(* PLC project contactor, Dassault Systèmes ControlBuild 2024x *)
(* stored: creationDateTime 2023-10-03T11:13:14-01:00 *)

(* This module simulates the interlocking of a contactor. It returns its state and a contactor feed-back. *)
FUNCTION_BLOCK equipment_library.contactor
  VAR_INPUT
    voltage380 : BOOL := true;
    cmdSupply : BOOL := true;
    sensorSupply : BOOL := true;
  END_VAR
  VAR_INPUT
    forward : BOOL := false;
  END_VAR
  VAR_OUTPUT
    forwardState : BOOL := false;
  END_VAR
  VAR_OUTPUT
    contactorFB : BOOL := false;
    thermal : BOOL := true;
  END_VAR
  VAR
    memoForward : BOOL := false;
  END_VAR
  VAR CONSTANT
    forwardLogic : BOOL := true;
    thermalLogic : BOOL := false;
  END_VAR
  VAR
    d_forward : BOOL := false;
    v_d_forward : BOOL := false;
    d_electrical : BOOL := false;
    v_d_electrical : BOOL := false;
  END_VAR


ACTION C_source_code:
/* ----------------------------------------------------------------	*/
/* Type : Model of Operative Behaviour					*/
/* Category :  Pre-actuators						*/
/* Author : Dassault Systemes						*/
/* Update date : June 2018							*/
/* ----------------------------------------------------------------	*/
/* This module simulates the interlocking of a contactor.  		*/
/* It returns its state and a contactor feed-back.			*/
/* ----------------------------------------------------------------	*/

/* ----------------------------------------------------------------	*/
/* Management of orders from Control Part					*/
/*	if there is no power supply for command 				*/
/*         the contactor doesn't understand the control order		*/
/* ----------------------------------------------------------------	*/
memoForward=forward & cmdSupply & ! d_electrical;

/* ----------------------------------------------------------------	*/
/* Calculation of the on-state of contactor				*/
/* ----------------------------------------------------------------	*/
forwardState=memoForward & voltage380;

/* ----------------------------------------------------------------	*/
/* Management of the thermal feed-back					*/
/* ----------------------------------------------------------------	*/
if (d_electrical) thermal = v_d_electrical;
else
	thermal = ! thermalLogic & sensorSupply;

/* ----------------------------------------------------------------	*/
/* Management of feedback to Control Part					*/
/*     if a fault is required, the contactor feed-back 		*/
/*		 takes a preset state.					*/
/*	if there is no power supply for sensor 				*/
/*         contactor feed-back returns nothing				*/
/*     else contactor feed-back returns the contactor state combined	*/
/*	    with wiring logic.						*/
/* ----------------------------------------------------------------	*/

if (d_forward) contactorFB = v_d_forward;
else
	contactorFB = (memoForward ^ ! forwardLogic) && sensorSupply;
END_ACTION
END_FUNCTION_BLOCK
